{attribute 'linkalways'} 
{attribute 'no_explicit_call' := 'This FB is a CLASS and must be accessed using methods or properties'}
{attribute 'enable_dynamic_creation'}
FUNCTION_BLOCK FINAL ADD_DINT EXTENDS Node
VAR
	in1 : _DINT(0);
	in2 : _DINT(0);
	out : _DINT(0);
END_VAR

METHOD PUBLIC Clone : I_Node
VAR
	pNode : POINTER TO ADD_DINT;
END_VAR
pNode := __NEW(ADD_DINT);
Clone := pNode^;
END_METHOD

METHOD FB_init : BOOL
VAR_INPUT
	bInitRetains : BOOL; // if TRUE, the retain variables are initialized (warm start / cold start)
	bInCopyCode : BOOL;  // if TRUE, the instance afterwards gets moved into the copy code (online change)
END_VAR
AddInput('in1',THIS^.in1);
AddInput('in2',THIS^.in2);
AddOutput('out', THIS^.out);
END_METHOD

METHOD PROTECTED OnExecute
VAR
END_VAR
out.Value := in1.Value + in2.Value;
END_METHOD

END_FUNCTION_BLOCK

(* stored: Version 1.1.0.1, ProductVersion 3.1.4024.15
   POU ADD_DINT: Id {ef7ac5a4-82a3-4959-9f10-bac8faf12740}, SpecialFunc None
   Folder Constructor: Id {588a486f-6871-4576-aee0-cbfc192f5dfa}
   Method Clone: Id {ee8790f2-c4f4-4ac5-bdae-9df049af4baa}
   Method FB_init: Id {071c9544-68b5-49f0-b9be-d57b6963a4ef}
   Method OnExecute: Id {adc6cc75-93ed-4de4-9a05-a748f346878c} *)
